// TIA Portal V21 export
VAR_GLOBAL   // PLC tag table "KAllAnalog"
END_VAR
VAR_GLOBAL CONSTANT   // user constants
   KAllAnalog_Maxi : Int := 1;
   KAllAnalog_IntMax : Int := 2;
   KAllAnalog_IntMin : Int := 3;
   KAllAnalog_Mini : Int := 4;
   KAllAnalog_OutOfRange : Int := 5;
END_VAR
